{attribute 'qualified_only'}
{attribute 'to_string'}
TYPE E_SelftestStates :
(
	Idle:=0,
	HomeStepper1,
	HomeStepper2,
	HomeLinearActuator1,
	HomeLinearActuator2,
	SetupEncoders1,
	SetupEncoders2,
	CheckAbsEncoderOffsets1,
	CheckAbsEncoderOffsets2,
	WrapUp
)UINT := Idle
;
END_TYPE

(* stored: Version 1.1.0.1, ProductVersion 3.1.4024.12
   EnumerationTextList E_SelftestStates: Id {01d4dc09-94db-4d4b-90b1-25185fe7eff3} *)
